(*
SPDX-FileCopyrightText: © 2026 Oleksandr Tiutyk <trofimich@gmail.com>
SPDX-License-Identifier: MIT
License: https://opensource.org/license/mit
*)

(*!
<summary>Runs the intersection and workflow samples through the automation runner.</summary>
<description>
Installs the sample log filter once before the first runner call, using local initialization state independent
of the system task cycle counter.
</description>
*)

PROGRAM MAIN
VAR_OUTPUT
	IntersectionHMI : HmiIntersectionController;
END_VAR
VAR
	{attribute 'hide'} 
	_IntersectionPlugings : ARRAY [0..0] OF TOF_Automation.IAutomationControllerPlugin := [IntersectionHMI];
END_VAR
VAR_OUTPUT	
	IntersectionController : IntersectionController("IntersectionController", _IntersectionPlugings);	
	DemoWorkflowController : DemoWorkflowController("DemoWorkflowController");
END_VAR
VAR
	{attribute 'hide'} 
	_AutomationControllers : ARRAY [0..1] OF TOF_Automation.IAutomationComponent := 
	[
		IntersectionController,
		DemoWorkflowController
	];
	
	{attribute 'hide'} 
	_LogFilter : LogFilter;
	{attribute 'hide'}
	_LogFilterInitialized : BOOL;
END_VAR
VAR_OUTPUT
	Runner : TOF_Automation.AutomationRunner(components := _AutomationControllers);
END_VAR

IF NOT _LogFilterInitialized THEN
	TOF_Core.LogManager.Filter := _LogFilter;
	_LogFilterInitialized := TRUE;
END_IF

Runner.Execute();

END_PROGRAM

(* stored: Version 1.1.0.1
   POU MAIN: Id {24d6dde4-f5e9-4d1b-910b-08a2682c02b5}, SpecialFunc None *)
